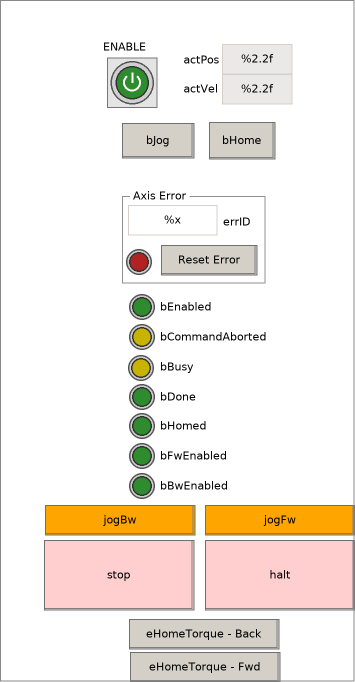
VISUALIZATION Torque  // 355x682
    GroupBox (122,188 143x95), "Axis Error"
    Button (209,122 66x37), "bHome"
        toggle HomeByTorque.bHome
    Button (122,123 72x35), "bJog"
        OnMouseDown: execute { HomeByTorque.bJog := TRUE; }
        OnMouseUp: execute { HomeByTorque.bJog := FALSE; }
    Lamp1 (124,247 30x30), variable: GVL.astAxes[3].stStatus.bError, style: Lamp-Lamp1-Red
    Button (161,245 96x30), "Reset Error", pressed state: GVL.astAxes[3].stControl.bReset, text list: 'languageTable', text index: "reset"
        OnMouseClick: toggle GVL.astAxes[3].stControl.bReset
    Textfield (128,205 89x30), "%x", text variable: GVL.astAxes[3].stStatus.nErrorID
    Textfield (220,207 44x30), "errID", text list: 'languageTable', text index: "errID"
    Textfield (157,471 117x30), "bBwEnabled", text list: 'languageTable', text index: "bBwEnabled"
    Lamp1 (127,292 30x30), variable: GVL.astAxes[3].stStatus.bEnabled, style: Lamp-Lamp1-Green
    Textfield (157,292 117x30), "bEnabled", text list: 'languageTable', text index: "bEnabled"
    Lamp1 (127,322 30x30), variable: GVL.astAxes[3].stStatus.bCommandAborted, style: Lamp-Lamp1-Yellow
    Textfield (157,322 117x30), "bCommandAborted", text list: 'languageTable', text index: "bCommandAborted"
    Textfield (157,352 117x30), "bBusy", text list: 'languageTable', text index: "bBusy"
    Lamp1 (127,382 30x30), variable: GVL.astAxes[3].stStatus.bDone, style: Lamp-Lamp1-Green
    Textfield (157,382 117x30), "bDone", text list: 'languageTable', text index: "bDone"
    Lamp1 (127,411 30x30), variable: GVL.astAxes[3].stStatus.bHomed, style: Lamp-Lamp1-Green
    Textfield (157,411 117x30), "bHomed", text list: 'languageTable', text index: "bHomed"
    Lamp1 (127,441 30x30), variable: GVL.astAxes[3].stStatus.bFwEnabled AND NOT GVL.astAxes[3].stStatus.bInterlockedFwd, style: Lamp-Lamp1-Green
    Lamp1 (127,471 30x30), variable: GVL.astAxes[3].stStatus.bBwEnabled AND NOT GVL.astAxes[3].stStatus.bInterlockedBwd, style: Lamp-Lamp1-Green
    Textfield (157,441 117x30), "bFwEnabled", text list: 'languageTable', text index: "bFwEnabled"
    Lamp1 (126,353 30x30), variable: GVL.astAxes[3].stStatus.bBusy, style: Lamp-Lamp1-Yellow
    Textfield (222,44 70x30), "%2.2f", text variable: GVL.astAxes[3].stStatus.fActPosition
    Textfield (168,45 54x30), "actPos", text list: 'languageTable', text index: "actposition"
    Textfield (172,74 49x30), "actVel", text list: 'languageTable', text index: "actVelocity"
    Textfield (222,74 70x30), "%2.2f", text variable: GVL.astAxes[3].stStatus.fActVelocity
    Textfield (100,34 92x26), "ENABLE", text list: 'languageSupport', text index: "enable"
    PowerSwitch (107,56 50x53), variable: GVL.astAxes[3].stControl.bEnable, behaviour: TOGGLE, style: Switch-PowerSwitch-Green
    Button (45,505 150x30), "jogBw", text list: "languageSupport", text index: "jogBw"
        OnMouseUp: execute { GVL.astAxes[3].stControl.bJogBwd:= FALSE; }
        OnMouseClick: execute {  }
        OnMouseDown: execute { GVL.astAxes[3].stControl.eCommand:=E_MotionFunctions.eJog; GVL.astAxes[3].stControl.bJogBwd:= TRUE; }
    Button (205,505 150x30), "jogFw", text list: "languageSupport", text index: "jogFw"
        OnMouseUp: execute { GVL.astAxes[3].stControl.bJogFwd:= FALSE; }
        OnMouseClick: execute {  }
        OnMouseDown: execute { GVL.astAxes[3].stControl.eCommand:=E_MotionFunctions.eJog; GVL.astAxes[3].stControl.bJogFwd:= TRUE; }
    Button (205,540 150x70), "halt", pressed state: GVL.astAxes[3].stControl.bHalt, input disabled if: GVL.astAxes[3].stStatus.bGeared, text list: "languageSupport", text index: "halt"
        toggle GVL.astAxes[3].stControl.bHalt
    Button (44,540 150x70), "stop", pressed state: GVL.astAxes[3].stControl.bStop, input disabled if: GVL.astAxes[3].stStatus.bGeared, text list: "languageSupport", text index: "stop"
        toggle GVL.astAxes[3].stControl.bStop
    Button (129,619 150x30), "eHomeTorque - Back", input disabled if: GVL.astAxes[3].stStatus.bGeared
        OnMouseClick: execute {
            GVL.astAxes[3].stControl.eCommand:=E_MotionFunctions.eHome;
            GVL.astAxes[3].stConfig.eHomeSeq:=E_HomingRoutines.eHomeToBlock_Bwd;
            GVL.astAxes[3].stControl.bExecute:=TRUE;
        }
    Button (130,652 150x30), "eHomeTorque - Fwd", input disabled if: GVL.astAxes[3].stStatus.bGeared
        OnMouseClick: execute {
            GVL.astAxes[3].stControl.eCommand:=E_MotionFunctions.eHome;
            GVL.astAxes[3].stConfig.eHomeSeq:=E_HomingRoutines.eHomeToBlock_Fwd;
            GVL.astAxes[3].stControl.bExecute:=TRUE;
        }
END_VISUALIZATION

(* stored: Version 1.1.0.1, ProductVersion 3.1.4024.10
   Visu Torque: Id {1797c93a-675d-4e62-80f4-c8cc8fe9d099} *)
